// TIA Portal V19 export
TYPE "LAF_typeUnitConfiguration"
// General configuration of the unit
// stored: Access Published
   STRUCT
      referenceDesignator { S7_SetPoint := 'True'} : "LAF_typeReferenceConfiguration";   // Configuration of the Reference Designators
   END_STRUCT;
END_TYPE
